// TIA Portal V19 export
FUNCTION_BLOCK "RT"   // FB1192, LAD
TITLE = Torsteuerung
{ S7_Optimized_Access := 'TRUE' }
// stored: AutoNumber false, MemoryReserve 100, SetENOAutomatically true
   VAR RETAIN
      In { ExternalAccessible := 'False'; ExternalVisible := 'False'; ExternalWritable := 'False'} : Struct
         NotHalt : Bool;
         MSS_ok : Bool;
         ok : Bool;
         Knauf_Auto : Bool;
         T_auf : Bool;   // Paneltaste
         T_zu : Bool;   // Paneltaste
         S_auf : Bool;
         S_zu : Bool;
         ErrQ : Bool;   // Fehlerquittung
         Sperrluft_ok : Bool;
         Kein_Gas_Alarm : Bool;
      END_STRUCT;
      Param { ExternalAccessible := 'False'; ExternalVisible := 'False'; ExternalWritable := 'False'} : Struct
         "TO" : Time := T#3s500ms;
      END_STRUCT;
      Zst { ExternalAccessible := 'False'; ExternalVisible := 'False'; ExternalWritable := 'False'} : Struct
         Req_Auf : Bool;
         Fehler : Bool;
         Sperre_QF : Bool;
         QF_sicher : Bool;
      END_STRUCT;
      Out { ExternalAccessible := 'False'; ExternalVisible := 'False'; ExternalWritable := 'False'} : Struct
         auf : Bool;
         zu : Bool;
      END_STRUCT;
      Mld { ExternalAccessible := 'False'; ExternalVisible := 'False'; ExternalWritable := 'False'} : Struct
         n_Auto : Bool;
         TO_auf : Bool;
         TO_zu : Bool;
         MSS : Bool;
         nok : Bool;
      END_STRUCT;
   END_VAR
   VAR
      IEC_Timer { ExternalAccessible := 'False'; ExternalVisible := 'False'; ExternalWritable := 'False'} : Struct
         TO_auf : TON_TIME;
         TO_zu : TON_TIME;
      END_STRUCT;
   END_VAR
   VAR_TEMP
      TO_auf : Bool;
      TO_zu : Bool;
   END_VAR
BEGIN

REGION Network 1 (SCL): Input
   // Panelbdienung und Sensoren --> Input()
   // Not-Halt
   #In.NotHalt := NOT "DB_PNOZ_IN_Out".In.NH_Frg_RT;
   // kein Gasalarm
   #In.Kein_Gas_Alarm :="E_Al_Gas_ok";
   // Sperrluftventilator an
   #In.Sperrluft_ok := "A_Frg_FU_Vent";

   // Schnittstelle zum Transportsystem
   #Zst.QF_sicher :=("E_S_Pos_BE_QF1" OR "E_S_Pos_Ue_QF1") AND ("E_S_Pos_BE_QF2" OR "E_S_Pos_Ue_QF2")
   AND NOT "A_Frg_FU_QF_WR02" AND NOT "A_Frg_FU_QF_WR03";
END_REGION

REGION Network 2 (SCL): Sammelstörung
   IF #In.ErrQ THEN
       #Zst.Fehler := FALSE;
   END_IF;
   IF #In.NotHalt OR NOT #In.MSS_ok OR NOT #In.ok OR #Mld.TO_auf OR #Mld.TO_zu THEN
       #Zst.Fehler := TRUE;
   END_IF;
END_REGION

REGION Network 3 (SCL): Ansteuerung
   IF NOT #Zst.Fehler AND #In.Kein_Gas_Alarm AND #In.Sperrluft_ok THEN
       IF #In.Knauf_Auto THEN
           // Automatikbetrieb
           IF #Zst.QF_sicher THEN
               #Out.auf := #Zst.Req_Auf;// wird von WR02/03 gebildet
               #Out.zu := NOT #Zst.Req_Auf;
           ELSE
               #Out.auf := FALSE;
               #Out.zu := FALSE;
           END_IF;
       ELSE
           // Handbetrieb
           IF #In.T_auf AND NOT #In.T_zu THEN
               #Out.auf := TRUE;
               #Out.zu := FALSE;
           END_IF;
           IF #In.T_zu AND NOT #In.T_auf AND #Zst.QF_sicher THEN
               #Out.zu := TRUE;
               #Out.auf := FALSE;
           END_IF;
       END_IF;
   ELSE // Not-Halt, n.i.O, MSS
       #Out.auf := FALSE;
       #Out.zu := FALSE;
   END_IF;

   // Endlagen erreicht
   IF #In.S_auf THEN
       #Out.auf := FALSE;
   END_IF;

   IF #In.S_zu THEN
       #Out.zu := FALSE;
   END_IF;
END_REGION

REGION Network 4 (SCL): Sperre
   // Fahrt WR02/03  verboten
   #Zst.Sperre_QF := NOT #In.S_auf OR #In.S_zu OR #Out.zu;
END_REGION

REGION Network 5 (SCL): Überwachung / Alarme
   // MSS / Zeitüberschreitung
   // nicht betriebsbereit
   #Mld.nok := NOT #In.ok AND NOT #In.NotHalt;
   // Motorschutzschalter
   #Mld.MSS := NOT #In.MSS_ok AND NOT #In.NotHalt;

   // nicht in Automatik
   #Mld.n_Auto := NOT #In.Knauf_Auto AND "DB_ANLAGE".BA.Automat_ein;

   // Zeitüberschreitung öffnen
   #IEC_Timer.TO_auf(IN := #Out.auf AND NOT #In.S_auf,
                        PT := #Param.TO,
                        Q => #TO_auf);
      IF #TO_auf THEN
          #Mld.TO_auf := TRUE;
      ELSIF #In.ErrQ THEN
          #Mld.TO_auf := FALSE;
      END_IF;
          // Zeitüberschreitung schließen
   #IEC_Timer.TO_zu(IN := #Out.zu AND NOT #In.S_zu,
                        PT := #Param.TO,
                        Q => #TO_zu);
       IF #TO_zu THEN
           #Mld.TO_zu := TRUE;
       ELSIF #In.ErrQ THEN
           #Mld.TO_zu := FALSE;
       END_IF;
END_REGION
END_FUNCTION_BLOCK
